// TIA Portal V20 export
TYPE "typeDevicesStatusSummary"
// General safety status of devices
// stored: Access Published, IsFailsafeCompliant true, Namespace Safety
   STRUCT
      allDevicesOk { ExternalWritable := 'False'} : Bool;   // All devices are released and acknowledged
      allEstopButtonsOK { ExternalWritable := 'False'} : Bool;   // All estop buttons are released and acknowledged
      allDoorsOK { ExternalWritable := 'False'} : Bool;   // All doors are released and acknowledged
      anyEstopButtonPressed { ExternalWritable := 'False'} : Bool;   // At least one estop button is pressed
      anyDoorOpen { ExternalWritable := 'False'} : Bool;   // At least one door is open
      anyDriveFault { ExternalWritable := 'False'} : Bool;   // At least one drive has a safety fault
      eStopDelayedOK { ExternalWritable := 'False'} : Bool;   // The delay estop OK signal is TRUE
      allZoneAutoSatrtOk { ExternalWritable := 'False'} : Bool;
   END_STRUCT;
END_TYPE
